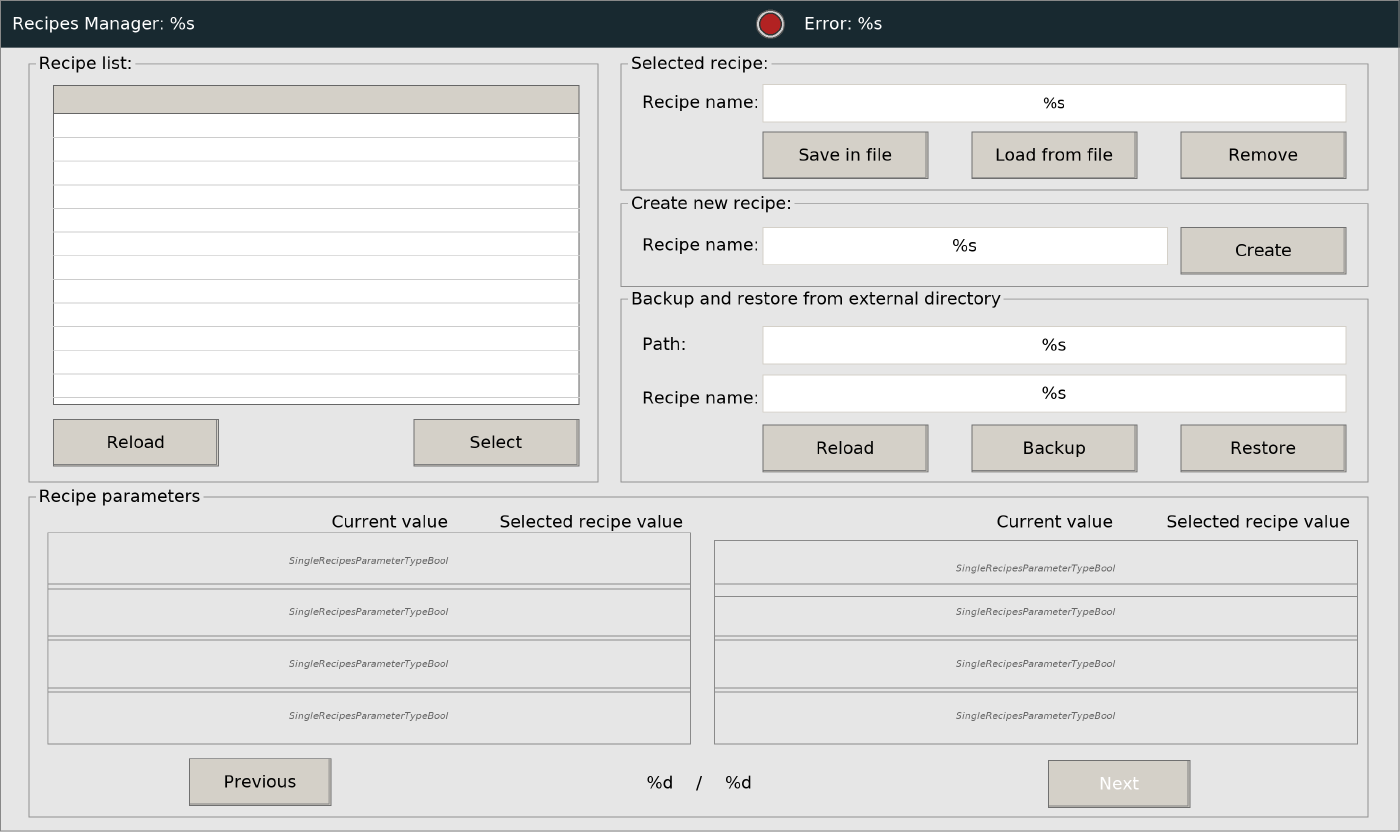
VISUALIZATION PageRecipesManager  // 1480x880
VAR_IN_OUT
	(* Recipe control - buttons *)
	btnCreate						: BOOL;						(* Create recipe button *)
	btnSelect						: BOOL;						(* Select recipe from table button*)
	btnLoad							: BOOL;						(* Load recipe from file button *)
	btnRead							: BOOL;						(* Read recipe to file button *)
	btnReload 						: BOOL;						(* Reload recipes button *)
	btnBackup						: BOOL;						(* Backup recipes to external directory button *)
	btnRestore						: BOOL;						(* Restore recipes from external directory button *)
	btnRecipeNext					: BOOL;						(* Go to next page with recipe parameters *)
	btnRecipePrevious				: BOOL;						(* Go to previous page with recipe parameters *)
	btnRemove						: BOOL;
	btnReloadExternal				: BOOL;
		
	(* Recipe control - visibility *)
	bReloadInvisible				: BOOL;						(* Makes reload button invisible *)
	bRecipeNextInvisible			: BOOL;						(* Makes next button invisible *)
	bRecipePreviousInvisible		: BOOL;						(* Makes previous button invisible *)
	bRecipeCreateInvisible			: BOOL;						(* Makes create group box invisible *)
	bRecipeBackupRestoreInvisible	: BOOL;						(* Makes backup and restore group box invisible *)
	bNoRecipeSelected				: BOOL;
	
	(* Recipe control - control disabled *)
	bRecipeCreateDisabled			: BOOL;						(* Disable access to create recipe group box *)
	bRecipeBackupRestoreDisabled	: BOOL;						(* Disable access to backup and restore group box *)
	
	(* Recipe control - status *)
	bError							: BOOL;						(* Error occured while executing last command *)
	eRecipesManagerReturns			: E_RecipesManagerReturns;	(* Result of last executed command *)
	eReacipeManagerState			: E_RecipesManagerState;	(* Current state of Recipe Manager *)
	
	(* Recipe control - parameters for recipes manager *)
	iSelectedRecipe					: INT;						(* Number of selected row in Available Recipes table *)
	sSelectedRecipe					: STRING;					(* Current selected recipe name - changes affter trigger from btnSelect *)
	sNewRecipeName					: STRING;					(* Name for new recipe *)
	sRestoreBackupPath				: STRING;				(* Path for backup/restoring of recipes *)
	sRestoreBackupRecipeName		: STRING;	
	arrRecipeNames					: ARRAY	[0..127] OF STRING;	(* Names of all detected recipes *)
	
	(* Recipe control - parameters data *)
	arrRecipeParameterFrameEmpty 	: ARRAY [0..7] OF BOOL;								(*  *)
	arrRecipeParameterFrameData		: ARRAY [0..7] OF ST_VisuCtrlRecipeParameter;		(*  *)
	arrRecipeParameterFrameType		: ARRAY [0..7] OF E_VisuCtrlRecipeParameterType;	(*  *)
	
	iRecipeSelectedPageIndex	: USINT;
	iRecipeTotalPageIndex 		: USINT;
END_VAR
    Rectangle (0,0 1480x50)
    Textfield (10,0 350x50), "Recipes Manager: %s", text list: 'TL_RecipesManagerStatus', text index: eReacipeManagerState
    GroupBox (30,517 1416x347), "Recipe parameters"
        Label (312,20 140x30), "Current value"
        Label (490,20 210x30), "Selected recipe value"
        Label (1010,20 150x30), "Current value"
        Label (1195,20 210x30), "Selected recipe value"
        Button (170,285 150x50), "Previous", invisible if: bRecipePreviousInvisible
            tap btnRecipePrevious
        Button (1078,287 150x50), "Next", invisible if: bRecipeNextInvisible
            tap btnRecipeNext
        Rectangle (644,286 130x50), "/"
        Rectangle (643,286 50x50), "%d", text variable: iRecipeSelectedPageIndex+1
        Rectangle (726,286 50x50), "%d", text variable: iRecipeTotalPageIndex+1
        Frame (20,100 680x60), invisible if: arrRecipeParameterFrameEmpty[1], frame switch variable: arrRecipeParameterFrameType[1]
            shows SingleRecipesParameterTypeBool(stRecipeParameter := arrRecipeParameterFrameData[1])
            shows SingleRecipesParameterTypeInteger(stRecipeParameter := arrRecipeParameterFrameData[1])
            shows SingleRecipesParameterTypeReal(stRecipeParameter := arrRecipeParameterFrameData[1])
            shows SingleRecipesParameterTypeString(stRecipeParameter := arrRecipeParameterFrameData[1])
        Frame (20,155 680x60), invisible if: arrRecipeParameterFrameEmpty[2], frame switch variable: arrRecipeParameterFrameType[2]
            shows SingleRecipesParameterTypeBool(stRecipeParameter := arrRecipeParameterFrameData[2])
            shows SingleRecipesParameterTypeInteger(stRecipeParameter := arrRecipeParameterFrameData[2])
            shows SingleRecipesParameterTypeReal(stRecipeParameter := arrRecipeParameterFrameData[2])
            shows SingleRecipesParameterTypeString(stRecipeParameter := arrRecipeParameterFrameData[2])
        Frame (20,210 680x60), invisible if: arrRecipeParameterFrameEmpty[3], frame switch variable: arrRecipeParameterFrameType[3]
            shows SingleRecipesParameterTypeBool(stRecipeParameter := arrRecipeParameterFrameData[3])
            shows SingleRecipesParameterTypeInteger(stRecipeParameter := arrRecipeParameterFrameData[3])
            shows SingleRecipesParameterTypeReal(stRecipeParameter := arrRecipeParameterFrameData[3])
            shows SingleRecipesParameterTypeString(stRecipeParameter := arrRecipeParameterFrameData[3])
        Frame (725,54 680x60), invisible if: arrRecipeParameterFrameEmpty[4], frame switch variable: arrRecipeParameterFrameType[4]
            shows SingleRecipesParameterTypeBool(stRecipeParameter := arrRecipeParameterFrameData[4])
            shows SingleRecipesParameterTypeInteger(stRecipeParameter := arrRecipeParameterFrameData[4])
            shows SingleRecipesParameterTypeReal(stRecipeParameter := arrRecipeParameterFrameData[4])
            shows SingleRecipesParameterTypeString(stRecipeParameter := arrRecipeParameterFrameData[4])
        Frame (725,100 680x60), invisible if: arrRecipeParameterFrameEmpty[5], frame switch variable: arrRecipeParameterFrameType[5]
            shows SingleRecipesParameterTypeBool(stRecipeParameter := arrRecipeParameterFrameData[5])
            shows SingleRecipesParameterTypeInteger(stRecipeParameter := arrRecipeParameterFrameData[5])
            shows SingleRecipesParameterTypeReal(stRecipeParameter := arrRecipeParameterFrameData[5])
            shows SingleRecipesParameterTypeString(stRecipeParameter := arrRecipeParameterFrameData[5])
        Frame (725,155 680x60), invisible if: arrRecipeParameterFrameEmpty[6], frame switch variable: arrRecipeParameterFrameType[6]
            shows SingleRecipesParameterTypeBool(stRecipeParameter := arrRecipeParameterFrameData[6])
            shows SingleRecipesParameterTypeInteger(stRecipeParameter := arrRecipeParameterFrameData[6])
            shows SingleRecipesParameterTypeReal(stRecipeParameter := arrRecipeParameterFrameData[6])
            shows SingleRecipesParameterTypeString(stRecipeParameter := arrRecipeParameterFrameData[6])
        Frame (725,210 680x60), invisible if: arrRecipeParameterFrameEmpty[7], frame switch variable: arrRecipeParameterFrameType[7]
            shows SingleRecipesParameterTypeBool(stRecipeParameter := arrRecipeParameterFrameData[7])
            shows SingleRecipesParameterTypeInteger(stRecipeParameter := arrRecipeParameterFrameData[7])
            shows SingleRecipesParameterTypeReal(stRecipeParameter := arrRecipeParameterFrameData[7])
            shows SingleRecipesParameterTypeString(stRecipeParameter := arrRecipeParameterFrameData[7])
        Frame (20,46 680x60), invisible if: arrRecipeParameterFrameEmpty[0], frame switch variable: arrRecipeParameterFrameType[0]
            shows SingleRecipesParameterTypeBool(stRecipeParameter := arrRecipeParameterFrameData[0])
            shows SingleRecipesParameterTypeInteger(stRecipeParameter := arrRecipeParameterFrameData[0])
            shows SingleRecipesParameterTypeReal(stRecipeParameter := arrRecipeParameterFrameData[0])
            shows SingleRecipesParameterTypeString(stRecipeParameter := arrRecipeParameterFrameData[0])
    GroupBox (30,59 602x451), "Recipe list:", invisible if: bRecipeCreateInvisible, input disabled if: bRecipeCreateDisabled
        Button (26,384 175x50), "Reload", invisible if: bReloadInvisible
            tap btnReload
        Table (26,31 556x338), text list: '', data array: arrRecipeNames
            p1137915858: iSelectedRecipe
            p3854506369: arrRecipeNames[INDEX]
            p2232123230: Available Recipes
        Button (407,384 175x50), "Select"
            tap btnSelect
    GroupBox (656,308 790x202), "Backup and restore from external directory"
        Button (371,141 175x50), "Backup"
            tap btnBackup
        Button (592,141 175x50), "Restore"
            tap btnRestore
        Textfield (150,37 617x40), "%s", text variable: sRestoreBackupPath
            OnMouseClick: write the text variable via VisuDialogs.Keypad
        Label (20,41 150x30), "Path:"
        Textfield (150,88 617x40), "%s", text variable: sRestoreBackupRecipeName
            OnMouseClick: write the text variable via VisuDialogs.Keypad
        Button (150,141 175x50), "Reload"
            tap btnReloadExternal
        Label (20,98 123x30), "Recipe name:"
    GroupBox (656,207 790x96), "Create new recipe:", invisible if: bRecipeCreateInvisible, input disabled if: bRecipeCreateDisabled
        Button (592,33 175x50), "Create"
            tap btnCreate
        Textfield (150,33 428x40), "%s", text variable: sNewRecipeName
            OnMouseClick: write the text variable via VisuDialogs.Keypad
        Label (20,37 150x30), "Recipe name:"
    GroupBox (656,59 790x142), "Selected recipe:", input disabled if: bNoRecipeSelected
        Button (150,80 175x50), "Save in file"
            tap btnRead
        Button (592,80 175x50), "Remove"
            tap btnRemove
        Textfield (150,30 617x40), "%s", text variable: sSelectedRecipe
        Button (371,80 175x50), "Load from file"
            tap btnLoad
        Label (20,34 150x30), "Recipe name:"
    Textfield (847,0 594x50), "Error: %s", text list: 'TL_RecipesManagerReturns', text index: eRecipesManagerReturns
    Lamp1 (797,8 35x35), variable: bError, style: Lamp-Lamp1-Red
END_VISUALIZATION

(* stored: Version 1.1.0.1, ProductVersion 3.1.4024.12
   Visu PageRecipesManager: Id {c2ffeee8-3e74-4505-af9e-b9cad1b8e443} *)
